// TIA Portal project "23Mayis" (V15)

(* hardware
DEVICE "S7-1200 station_1"  S7-1200 Station
   slot 0: "Rack_0"  S7-1200 Rack  Rack  V1.0
   slot 1: "PLC_1"  CPU 1214C DC/DC/DC  6ES7 214-1AG40-0XB0  V4.2
*)

// ===== PLC "PLC_1"  CPU 1214C DC/DC/DC =====

VAR_GLOBAL   // PLC tag table "Default tag table"
   "Sonuc_1" AT %MD0 : Real;
   "Sonuc_2" AT %MD4 : Real;
   "Sonuc_3" AT %MD8 : Real;
   "Sonuc_4" AT %MD12 : Real;
   "Sonuc_5" AT %MD16 : Real;
   "Sonuc_6" AT %MD20 : Real;
   "A" AT %MD24 : Real;
   "B" AT %MD28 : Real;
   "E" AT %MD32 : Real;
   "D" AT %MD36 : Real;
END_VAR

ORGANIZATION_BLOCK "Main"   // OB1, LAD, ProgramCycle
TITLE = "Main Program Sweep (Cycle)"
{ S7_Optimized_Access := 'TRUE' }
VERSION : 0.1
   VAR_INPUT
      Initial_Call : Bool;   // Initial call of this OB
      Remanence : Bool;   // =True, if remanent data are available
   END_VAR
BEGIN

REGION Network 1: Soru1
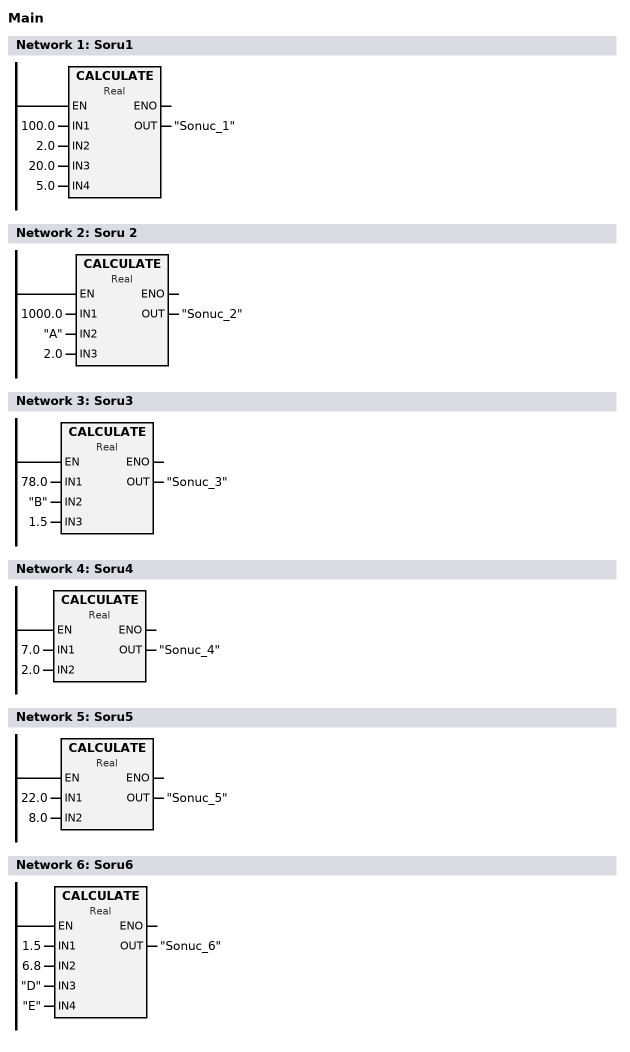
   RUNG wire#powerrail
      { S7_Templates := "SrcType := Real"; S7_Expression := "(IN1/IN2) + (IN3*IN4)-IN4" } Calculate(in1 := 100.0, in2 := 2.0, in3 := 20.0, in4 := 5.0, out => "Sonuc_1")
   END_RUNG
   // the same network as SCL:
   "Sonuc_1" := (100.0/2.0) + (20.0*5.0)-5.0;
END_REGION

REGION Network 2: Soru 2
   RUNG wire#powerrail
      { S7_Templates := "SrcType := Real"; S7_Expression := "(IN1*(IN2/IN3))" } Calculate(in1 := 1000.0, in2 := "A", in3 := 2.0, out => "Sonuc_2")
   END_RUNG
   // the same network as SCL:
   "Sonuc_2" := (1000.0*("A"/2.0));
END_REGION

REGION Network 3: Soru3
   RUNG wire#powerrail
      { S7_Templates := "SrcType := Real"; S7_Expression := "(IN1*(IN2*IN3))" } Calculate(in1 := 78.0, in2 := "B", in3 := 1.5, out => "Sonuc_3")
   END_RUNG
   // the same network as SCL:
   "Sonuc_3" := (78.0*("B"*1.5));
END_REGION

REGION Network 4: Soru4
   RUNG wire#powerrail
      { S7_Templates := "SrcType := Real"; S7_Expression := "IN1/IN2" } Calculate(in1 := 7.0, in2 := 2.0, out => "Sonuc_4")
   END_RUNG
   // the same network as SCL:
   "Sonuc_4" := 7.0/2.0;
END_REGION

REGION Network 5: Soru5
   RUNG wire#powerrail
      { S7_Templates := "SrcType := Real"; S7_Expression := "IN1/IN2" } Calculate(in1 := 22.0, in2 := 8.0, out => "Sonuc_5")
   END_RUNG
   // the same network as SCL:
   "Sonuc_5" := 22.0/8.0;
END_REGION

REGION Network 6: Soru6
   RUNG wire#powerrail
      { S7_Templates := "SrcType := Real"; S7_Expression := "IN1 + IN2 + (IN3*IN4)" } Calculate(in1 := 1.5, in2 := 6.8, in3 := "D", in4 := "E", out => "Sonuc_6")
   END_RUNG
   // the same network as SCL:
   "Sonuc_6" := 1.5 + 6.8 + ("D"*"E");
END_REGION
END_ORGANIZATION_BLOCK